{attribute 'linkalways'} 
{attribute 'no_explicit_call' := 'This FB is a CLASS and must be accessed using methods or properties'}
{attribute 'enable_dynamic_creation'}
FUNCTION_BLOCK FINAL NE_UINT EXTENDS Node
VAR
	in1 : _UINT(0);
	in2 : _UINT(0);
	out : _BOOL(FALSE);
END_VAR

METHOD PUBLIC Clone : I_Node
VAR
	pNode : POINTER TO NE_UINT;
END_VAR
pNode := __NEW(NE_UINT);
Clone := pNode^;
END_METHOD

METHOD FB_init : BOOL
VAR_INPUT
	bInitRetains : BOOL; // if TRUE, the retain variables are initialized (warm start / cold start)
	bInCopyCode : BOOL;  // if TRUE, the instance afterwards gets moved into the copy code (online change)
END_VAR
AddInput('in1',THIS^.in1);
AddInput('in2',THIS^.in2);
AddOutput('out', THIS^.out);
END_METHOD

METHOD PROTECTED OnExecute
VAR
END_VAR
out.Value := in1.Value <> in2.Value;
END_METHOD

END_FUNCTION_BLOCK

(* stored: Version 1.1.0.1, ProductVersion 3.1.4024.15
   POU NE_UINT: Id {b07b247b-3048-4a5f-8c15-8a2544d3a57b}, SpecialFunc None
   Folder Constructor: Id {765ad1d1-8415-41be-9b38-78361bc2718c}
   Method Clone: Id {ed442ac5-cc02-4bd7-ab74-029b53b56f02}
   Method FB_init: Id {4e802325-d139-492c-aa43-c0c4c68fc2ad}
   Method OnExecute: Id {5af5bb9e-5151-4f98-a228-874931ecfcf0} *)
